# EPICS substitutions: ek9000App/Db/EL3111.substitutions
file EL3111.template
{       pattern
        {
                TERMINAL,

        }
        {
        }
}
